TYPE SampleStruct :
STRUCT
	iNumericProperty: INT;
	sStringProperty: STRING;
END_STRUCT
END_TYPE

(* stored: Version 1.1.0.1, ProductVersion 3.1.4022.12
   DUT SampleStruct: Id {bd32e3b3-ac20-433b-98a6-be48d8ded8c6} *)
